# EPICS substitutions: apps/caenHvApp/Db/HVDCb_sums.substitutions
file "db/HVDC_sums.db" {
    pattern {S,R,L}
    {"4","1","1"}
    {"4","1","2"}
    {"4","2","3"}
    {"4","2","4"}
    {"4","3","5"}
    {"4","3","6"}
    {"5","1","1"}
    {"5","1","2"}
    {"5","2","3"}
    {"5","2","4"}
    {"5","3","5"}
    {"5","3","6"}
    {"6","1","1"}
    {"6","1","2"}
    {"6","2","3"}
    {"6","2","4"}
    {"6","3","5"}
    {"6","3","6"}
}
